// TIA Portal V20 export
DATA_BLOCK "process_DB_1"   // DB4
// stored: InstanceOfName ELY_1.process, InstanceOfType FB, Namespace ELY_1
"ELY_1.process"
   // VAR_INPUT
   //    Done : Bool;
   // END_VAR
BEGIN
END_DATA_BLOCK
